// TIA Portal project "myproject" (V16)

(* hardware
DEVICE "S71500/ET200MP-Station_1"  S7-1500 station
   slot 0: "Profilschiene_0"  6ES7 590-1***0-0AA0
   slot 1: "PLC_1"  CPU 1511-1 PN  6ES7 511-1AK00-0AB0  V1.8
   slot 2: "AI 8xU/I/RTD/TC ST_1"  AI 8xU/I/RTD/TC ST  6ES7 531-7KF00-0AB0  V2.0
   slot 3: "AI 8xU/I/RTD/TC ST_2"  AI 8xU/I/RTD/TC ST  6ES7 531-7KF00-0AB0  V2.0
   slot 4: "AI 8xU/I/RTD/TC ST_3"  AI 8xU/I/RTD/TC ST  6ES7 531-7KF00-0AB0  V2.0
   slot 5: "AI 8xU/I/RTD/TC ST_4"  AI 8xU/I/RTD/TC ST  6ES7 531-7KF00-0AB0  V2.0
   slot 6: "DI 16x24VDC BA_1"  DI 16x24VDC BA  6ES7 521-1BH10-0AA0  V1.0
   slot 7: "DI 16x24VDC / DQ 16x24VDC/0.5A BA_1"  DI 16x24VDC/DQ 16x24VDC/0.5A BA  6ES7 523-1BL00-0AA0  V1.1
   slot 8: "DI 16x24VDC / DQ 16x24VDC/0.5A BA_2"  DI 16x24VDC/DQ 16x24VDC/0.5A BA  6ES7 523-1BL00-0AA0  V1.1
DEVICE "HMI_1"  TP700 Comfort INOX PCT
   slot 0: "HMI_1"  TP700 Comfort INOX PCT  6AV2 144-8GC20-0AA0  16.0.0.0
   slot 1: "HMI_RT_1"  TP700 Comfort INOX PCT  6AV2 144-8GC20-0AA0  16.0.0.0
   slot 5: "HMI_1.IE_CP_1"  PROFINET Interface  16.0.0.0
      slot 1: "PROFINET Interface_1"  PROFINET Interface
         slot 1: "Port_1"  Port
         slot 2: "Port_2"  Port
   slot 7: "HMI_1.MPI/DP_CP_1"  MPI/DP Interface  16.0.0.0
*)

// ===== PLC "PLC_1"  CPU 1511-1 PN =====

VAR_GLOBAL   // PLC tag table "Standard-Variablentabelle"
   "compteur_boites" AT %C1 : Counter;
   "compteur_bouteilles" AT %C2 : Counter;
   "tag11" AT %M6.1 : Bool;
END_VAR

VAR_GLOBAL   // PLC tag table "Input/output"
   "c1" AT %I0.0 : Bool;   // capteur plastique fondu
   "mc1" AT %Q0.0 : Bool;   // moteur convoyeur 1
   "cm1" AT %I0.1 : Bool;   // capteur devant machine 1
   "m1" AT %Q0.1 : Bool;   // moteur machine moulage
   "cm11" AT %I0.2 : Bool;   // capteur apres machine moulage
   "mc2" AT %Q0.2 : Bool;   // moteur convoyeur 2
   "mcb" AT %Q0.3 : Bool;   // moteur curved belt
   "cl" AT %I0.3 : Bool;   // capteur boite
   "lids conveyor" AT %Q0.4 : Bool;   // convoyeur boite-assemblage
   "base conveyor" AT %Q0.5 : Bool;   // convoyeur base-assemblage
   "lid clamped" AT %I0.4 : Bool;   // clamped boite
   "base clamped" AT %I0.5 : Bool;   // clamped base
   "clamp lid" AT %Q0.6 : Bool;   // clamper la boite
   "clamp base" AT %Q0.7 : Bool;   // clamper la base
   "move x assemb" AT %Q1.0 : Bool;   // translation m. assemblage sur x
   "move z assemb" AT %Q1.1 : Bool;   // translation m. assemblage sur z
   "moved x assemb" AT %I0.6 : Bool;   // translation en cours sur x
   "moved z assemb" AT %I0.7 : Bool;   // translation en cours sur z
   "raise assemb" AT %Q1.2 : Bool;   // relever la barre devant produit assemblé
   "grab assemb" AT %Q1.3 : Bool;   // grab de la boite
   "grabbed assemb" AT %I1.4 : Bool;   // boite grabbed
   "lid at place" AT %I1.0 : Bool;   // boite en place
   "base at place" AT %I1.1 : Bool;   // base en place
   "part leaving" AT %I1.2 : Bool;   // piece sortante
   "cc" AT %I1.3 : Bool;   // capteur bol
   "ettiquetage conveyor" AT %Q1.5 : Bool;   // convoyeur ettiquette
   "product conveyor" AT %Q1.6 : Bool;   // convoyeur bol/ettiquetage
   "box clamped" AT %I2.7 : Bool;   // clamped ett
   "product clamped" AT %I1.5 : Bool;   // clamped bol/ettiquetage
   "clamp ettiquete" AT %Q1.7 : Bool;   // clamper l'ettiquette
   "clamp product" AT %Q2.0 : Bool;   // clamper le bol/ettiquetage
   "move x ett" AT %Q2.1 : Bool;   // translation m. etti sur x
   "move z ett" AT %Q2.2 : Bool;   // translation m. etti sur z
   "moved x ett" AT %I1.6 : Bool;   // translation en cours sur x
   "moved z ett" AT %I1.7 : Bool;   // translation en cours sur z
   "raise ett" AT %Q2.3 : Bool;   // relever la barre devant produit etti
   "grab ett" AT %Q2.4 : Bool;   // grab du produit
   "grabbed ett" AT %I3.1 : Bool;   // produit grabbed
   "ettiquete at place" AT %I2.0 : Bool;   // ettiquete en place
   "product at place" AT %I2.1 : Bool;   // produit en place
   "product leaving" AT %I2.2 : Bool;   // produit sortant
   "dcy" AT %I2.3 : Bool;   // bouton debut cycle
   "fcy" AT %I2.4 : Bool;   // bouton fin cycle
   "au" AT %I2.5 : Bool;   // bouton urgence
   "emetteur plastique" AT %Q2.6 : Bool;   // emetteur plastique fondu
   "emetteur base" AT %Q2.7 : Bool;   // emetteur base du jouet
   "emetteur bol" AT %Q3.0 : Bool;   // emetteur carton d'emballage
   "emetteur ettiquete" AT %Q3.1 : Bool;   // emetteur box d'emballage
   "tag1" AT %M3.2 : Bool;
   "tag2" AT %M3.3 : Bool;
   "tag3" AT %M3.4 : Bool;
   "tag4" AT %M3.5 : Bool;
   "cp" AT %I3.0 : Bool;   // capteur piece assemblée
   "raised assembly" AT %I3.2 : Bool;   // barre raised assembly
   "raised ettiq" AT %I3.3 : Bool;   // barre raised ett
   "bol conveyor" AT %Q3.2 : Bool;   // convoyeur des bols
   "cp2" AT %I3.4 : Bool;   // capteur piece assemblée sortante
   "cb" AT %I3.5 : Bool;   // capteur ettiquette
   "cp3" AT %I3.6 : Bool;   // capteur produit ettiqueté
   "tag5" AT %M3.7 : Bool;
   "tag6" AT %M4.0 : Bool;
   "tag7" AT %M4.1 : Bool;
   "tag8" AT %M4.2 : Bool;
   "remover" AT %Q3.3 : Bool;   // stock de sortie
   "tag9" AT %M5.7 : Bool;
   "vv" AT %Q3.4 : Bool;   // voyant vert de marche du systeme
   "vo" AT %Q3.5 : Bool;   // voyant orangé d'arret fin de cycle
   "vr" AT %Q3.6 : Bool;   // voyant rouge d'arret d'urgence
   "tag10" AT %M6.0 : Bool;
END_VAR

// folder: System blocks/Program resources

DATA_BLOCK "tp move z"   // DB1
{ S7_Optimized_Access := 'TRUE' }
AUTHOR : Simatic
FAMILY : IEC
NAME : IEC_TMR
VERSION : 1.0
// stored: InstanceOfName IEC_TIMER
"IEC_TIMER"
BEGIN
END_DATA_BLOCK

DATA_BLOCK "timer3"   // DB2
{ S7_Optimized_Access := 'TRUE' }
AUTHOR : Simatic
FAMILY : IEC
NAME : IEC_TMR
VERSION : 1.0
// stored: InstanceOfName IEC_TIMER
"IEC_TIMER"
BEGIN
END_DATA_BLOCK

DATA_BLOCK "time1"   // DB3
{ S7_Optimized_Access := 'TRUE' }
AUTHOR : Simatic
FAMILY : IEC
NAME : IEC_TMR
VERSION : 1.0
// stored: InstanceOfName IEC_TIMER
"IEC_TIMER"
BEGIN
END_DATA_BLOCK

DATA_BLOCK "timer4"   // DB4
{ S7_Optimized_Access := 'TRUE' }
AUTHOR : Simatic
FAMILY : IEC
NAME : IEC_TMR
VERSION : 1.0
// stored: InstanceOfName IEC_TIMER
"IEC_TIMER"
BEGIN
END_DATA_BLOCK

DATA_BLOCK "counter_boites"   // DB5
{ S7_Optimized_Access := 'TRUE' }
AUTHOR : Simatic
FAMILY : IEC
NAME : CNTR
VERSION : 1.0
// stored: InstanceOfName IEC_COUNTER
"IEC_COUNTER"
BEGIN
END_DATA_BLOCK

DATA_BLOCK "counter_bols"   // DB6
{ S7_Optimized_Access := 'TRUE' }
AUTHOR : Simatic
FAMILY : IEC
NAME : CNTR
VERSION : 1.0
// stored: InstanceOfName IEC_COUNTER
"IEC_COUNTER"
BEGIN
END_DATA_BLOCK

// folder: (top level)

FUNCTION "MHJ-PLC-Lab-Function-S71500" : Void   // FC9000, SCL
{ S7_Optimized_Access := 'TRUE' }
VERSION : 0.1
   VAR_TEMP
      Value : Byte;
      ForCounter : Int;
   END_VAR
   VAR CONSTANT
      Value_01_DW : DWord := 16#1223_5486;
      Value_02_DW : DWord := 16#A6C9_D1F5;
   END_VAR
BEGIN

   #Value:=PEEK(area := 16#82,
        dbNumber := 0,
        byteOffset := 511);
   #Value := #Value + 1;

   POKE(area := 16#82,
        dbNumber := 0,
        byteOffset := 511,
        value := #Value);

   POKE(area := 16#82,
        dbNumber := 0,
        byteOffset := 1016,
        value := #Value_01_DW);
   POKE(area := 16#82,
        dbNumber := 0,
        byteOffset := 1020,
        value := #Value_02_DW);

   FOR #ForCounter := 0 TO 63 DO
       #Value:=PEEK(area := 16#1,
            dbNumber := 0,
            byteOffset := #ForCounter);
       POKE(area := 16#81,
            dbNumber := 0,
            byteOffset := #ForCounter,
            value := #Value);
   END_FOR;
   #Value := PEEK(area := 16#1,
                  dbNumber := 0,
                  byteOffset := 512);
   POKE(area := 16#82,
        dbNumber := 0,
        byteOffset := 512,
        value := #Value);
END_FUNCTION

ORGANIZATION_BLOCK "Main"   // OB1, LAD, ProgramCycle
TITLE = "Main Program Sweep (Cycle)"
{ S7_Optimized_Access := 'TRUE' }
VERSION : 0.1
   VAR_INPUT
      Initial_Call : Bool;   // Initial call of this OB
      Remanence : Bool;   // =True, if remanent data are available
   END_VAR
   VAR_TEMP   // added for the SCL form of the ladder/FBD networks
      _w1 : Bool;
      _w2 : Bool;
   END_VAR
BEGIN

REGION Network 1
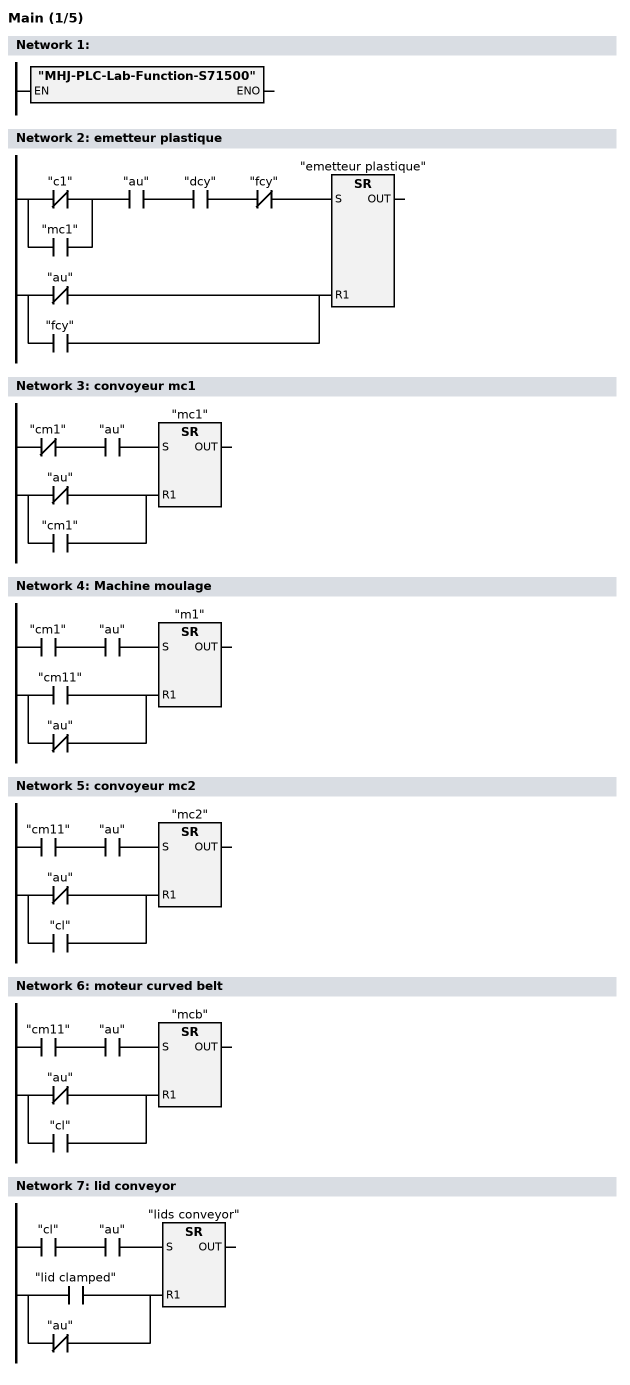
   RUNG wire#powerrail
      "MHJ-PLC-Lab-Function-S71500"()
   END_RUNG
   // the same network as SCL:
   "MHJ-PLC-Lab-Function-S71500"();
END_REGION

REGION Network 2: emetteur plastique
   RUNG wire#powerrail
      I_Contact( "c1" )
      wire#w1
      Contact( "au" )
      Contact( "dcy" )
      I_Contact( "fcy" )
      S_SR(operand := "emetteur plastique", r1 := wire#w2)
   END_RUNG
   RUNG wire#powerrail
      Contact( "mc1" )
   END_RUNG wire#w1
   RUNG wire#powerrail
      I_Contact( "au" )
   END_RUNG wire#w2
   RUNG wire#powerrail
      Contact( "fcy" )
   END_RUNG wire#w2
   // the same network as SCL:
   IF (NOT "c1" OR "mc1") AND "au" AND "dcy" AND NOT "fcy" THEN
       "emetteur plastique" := TRUE;   // SR flip-flop
   END_IF;
   IF NOT "au" OR "fcy" THEN "emetteur plastique" := FALSE; END_IF;
END_REGION

REGION Network 3: convoyeur mc1
   RUNG wire#powerrail
      I_Contact( "cm1" )
      Contact( "au" )
      S_SR(operand := "mc1", r1 := wire#w1)
   END_RUNG
   RUNG wire#powerrail
      I_Contact( "au" )
   END_RUNG wire#w1
   RUNG wire#powerrail
      Contact( "cm1" )
   END_RUNG wire#w1
   // the same network as SCL:
   IF NOT "cm1" AND "au" THEN
       "mc1" := TRUE;   // SR flip-flop
   END_IF;
   IF NOT "au" OR "cm1" THEN "mc1" := FALSE; END_IF;
END_REGION

REGION Network 4: Machine moulage
   RUNG wire#powerrail
      Contact( "cm1" )
      Contact( "au" )
      S_SR(operand := "m1", r1 := wire#w1)
   END_RUNG
   RUNG wire#powerrail
      Contact( "cm11" )
   END_RUNG wire#w1
   RUNG wire#powerrail
      I_Contact( "au" )
   END_RUNG wire#w1
   // the same network as SCL:
   IF "cm1" AND "au" THEN
       "m1" := TRUE;   // SR flip-flop
   END_IF;
   IF "cm11" OR NOT "au" THEN "m1" := FALSE; END_IF;
END_REGION

REGION Network 5: convoyeur mc2
   RUNG wire#powerrail
      Contact( "cm11" )
      Contact( "au" )
      S_SR(operand := "mc2", r1 := wire#w1)
   END_RUNG
   RUNG wire#powerrail
      I_Contact( "au" )
   END_RUNG wire#w1
   RUNG wire#powerrail
      Contact( "cl" )
   END_RUNG wire#w1
   // the same network as SCL:
   IF "cm11" AND "au" THEN
       "mc2" := TRUE;   // SR flip-flop
   END_IF;
   IF NOT "au" OR "cl" THEN "mc2" := FALSE; END_IF;
END_REGION

REGION Network 6: moteur curved belt
   RUNG wire#powerrail
      Contact( "cm11" )
      Contact( "au" )
      S_SR(operand := "mcb", r1 := wire#w1)
   END_RUNG
   RUNG wire#powerrail
      I_Contact( "au" )
   END_RUNG wire#w1
   RUNG wire#powerrail
      Contact( "cl" )
   END_RUNG wire#w1
   // the same network as SCL:
   IF "cm11" AND "au" THEN
       "mcb" := TRUE;   // SR flip-flop
   END_IF;
   IF NOT "au" OR "cl" THEN "mcb" := FALSE; END_IF;
END_REGION

REGION Network 7: lid conveyor
   RUNG wire#powerrail
      Contact( "cl" )
      Contact( "au" )
      S_SR(operand := "lids conveyor", r1 := wire#w1)
   END_RUNG
   RUNG wire#powerrail
      Contact( "lid clamped" )
   END_RUNG wire#w1
   RUNG wire#powerrail
      I_Contact( "au" )
   END_RUNG wire#w1
   // the same network as SCL:
   IF "cl" AND "au" THEN
       "lids conveyor" := TRUE;   // SR flip-flop
   END_IF;
   IF "lid clamped" OR NOT "au" THEN "lids conveyor" := FALSE; END_IF;
END_REGION

REGION Network 8: clamping lid
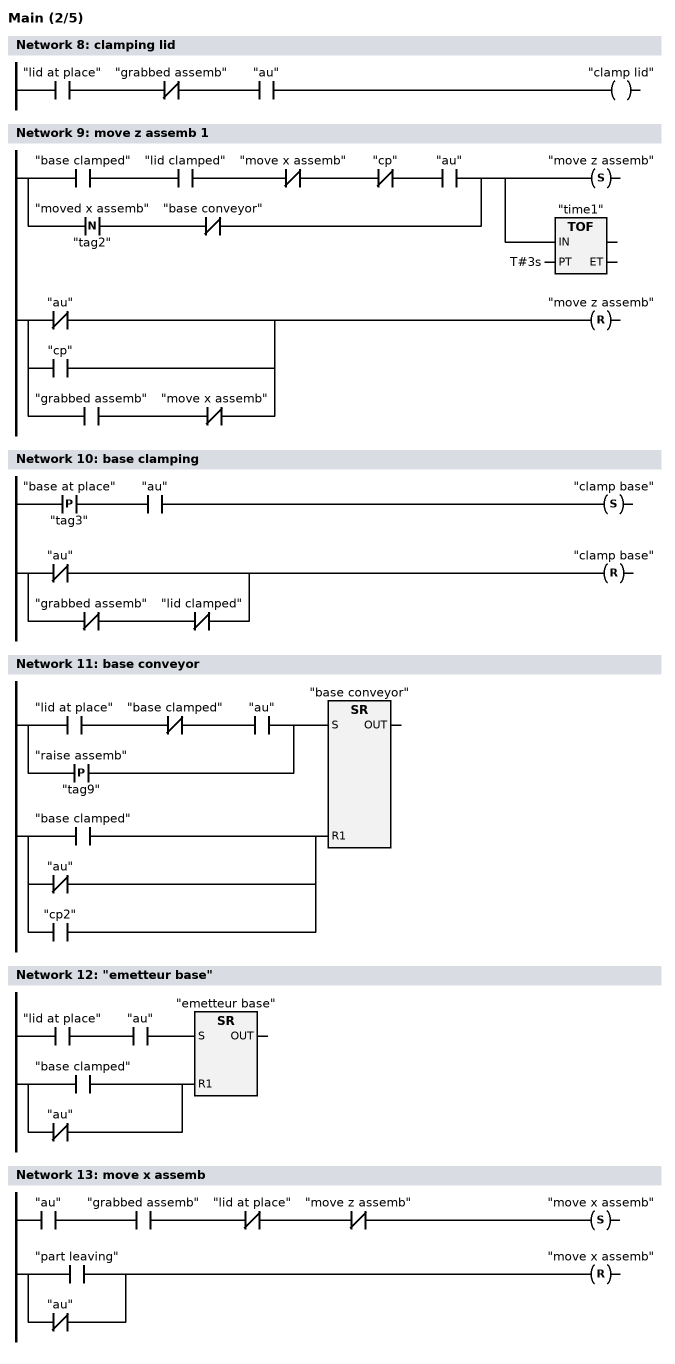
   RUNG wire#powerrail
      Contact( "lid at place" )
      I_Contact( "grabbed assemb" )
      Contact( "au" )
      Coil( "clamp lid" )
   END_RUNG
   // the same network as SCL:
   "clamp lid" := "lid at place" AND NOT "grabbed assemb" AND "au";
END_REGION

REGION Network 9: move z assemb 1
   #_w1 := NOT "moved x assemb" AND "tag2";   // falling edge of "moved x assemb"
   "tag2" := "moved x assemb";
   #_w2 := ("base clamped" AND "lid clamped" AND NOT "move x assemb" AND NOT "cp" AND "au") OR (#_w1 AND NOT "base conveyor");
   IF #_w2 THEN "move z assemb" := TRUE; END_IF;
   "time1".TOF(IN := #_w2, PT := T#3s);
   IF NOT "au" OR "cp" OR ("grabbed assemb" AND NOT "move x assemb") THEN "move z assemb" := FALSE; END_IF;
END_REGION

REGION Network 10: base clamping
   RUNG wire#powerrail
      P_Contact(operand := "base at place", bit := "tag3")
      Contact( "au" )
      S_Coil( "clamp base" )
   END_RUNG
   RUNG wire#powerrail
      I_Contact( "au" )
      wire#w1
      R_Coil( "clamp base" )
   END_RUNG
   RUNG wire#powerrail
      I_Contact( "grabbed assemb" )
      I_Contact( "lid clamped" )
   END_RUNG wire#w1
   // the same network as SCL:
   #_w1 := "base at place" AND NOT "tag3";   // rising edge of "base at place"
   "tag3" := "base at place";
   IF #_w1 AND "au" THEN "clamp base" := TRUE; END_IF;
   IF NOT "au" OR (NOT "grabbed assemb" AND NOT "lid clamped") THEN "clamp base" := FALSE; END_IF;
END_REGION

REGION Network 11: base conveyor
   RUNG wire#powerrail
      Contact( "lid at place" )
      I_Contact( "base clamped" )
      Contact( "au" )
      wire#w1
      S_SR(operand := "base conveyor", r1 := wire#w2)
   END_RUNG
   RUNG wire#powerrail
      P_Contact(operand := "raise assemb", bit := "tag9")
   END_RUNG wire#w1
   RUNG wire#powerrail
      Contact( "base clamped" )
   END_RUNG wire#w2
   RUNG wire#powerrail
      I_Contact( "au" )
   END_RUNG wire#w2
   RUNG wire#powerrail
      Contact( "cp2" )
   END_RUNG wire#w2
   // the same network as SCL:
   #_w1 := "raise assemb" AND NOT "tag9";   // rising edge of "raise assemb"
   "tag9" := "raise assemb";
   IF ("lid at place" AND NOT "base clamped" AND "au") OR #_w1 THEN
       "base conveyor" := TRUE;   // SR flip-flop
   END_IF;
   IF "base clamped" OR NOT "au" OR "cp2" THEN "base conveyor" := FALSE; END_IF;
END_REGION

REGION Network 12: "emetteur base"
   RUNG wire#powerrail
      Contact( "lid at place" )
      Contact( "au" )
      S_SR(operand := "emetteur base", r1 := wire#w1)
   END_RUNG
   RUNG wire#powerrail
      Contact( "base clamped" )
   END_RUNG wire#w1
   RUNG wire#powerrail
      I_Contact( "au" )
   END_RUNG wire#w1
   // the same network as SCL:
   IF "lid at place" AND "au" THEN
       "emetteur base" := TRUE;   // SR flip-flop
   END_IF;
   IF "base clamped" OR NOT "au" THEN "emetteur base" := FALSE; END_IF;
END_REGION

REGION Network 13: move x assemb
   RUNG wire#powerrail
      Contact( "au" )
      Contact( "grabbed assemb" )
      I_Contact( "lid at place" )
      I_Contact( "move z assemb" )
      S_Coil( "move x assemb" )
   END_RUNG
   RUNG wire#powerrail
      Contact( "part leaving" )
      wire#w1
      R_Coil( "move x assemb" )
   END_RUNG
   RUNG wire#powerrail
      I_Contact( "au" )
   END_RUNG wire#w1
   // the same network as SCL:
   IF "au" AND "grabbed assemb" AND NOT "lid at place" AND NOT "move z assemb" THEN
       "move x assemb" := TRUE;
   END_IF;
   IF "part leaving" OR NOT "au" THEN "move x assemb" := FALSE; END_IF;
END_REGION

REGION Network 14: grab assem
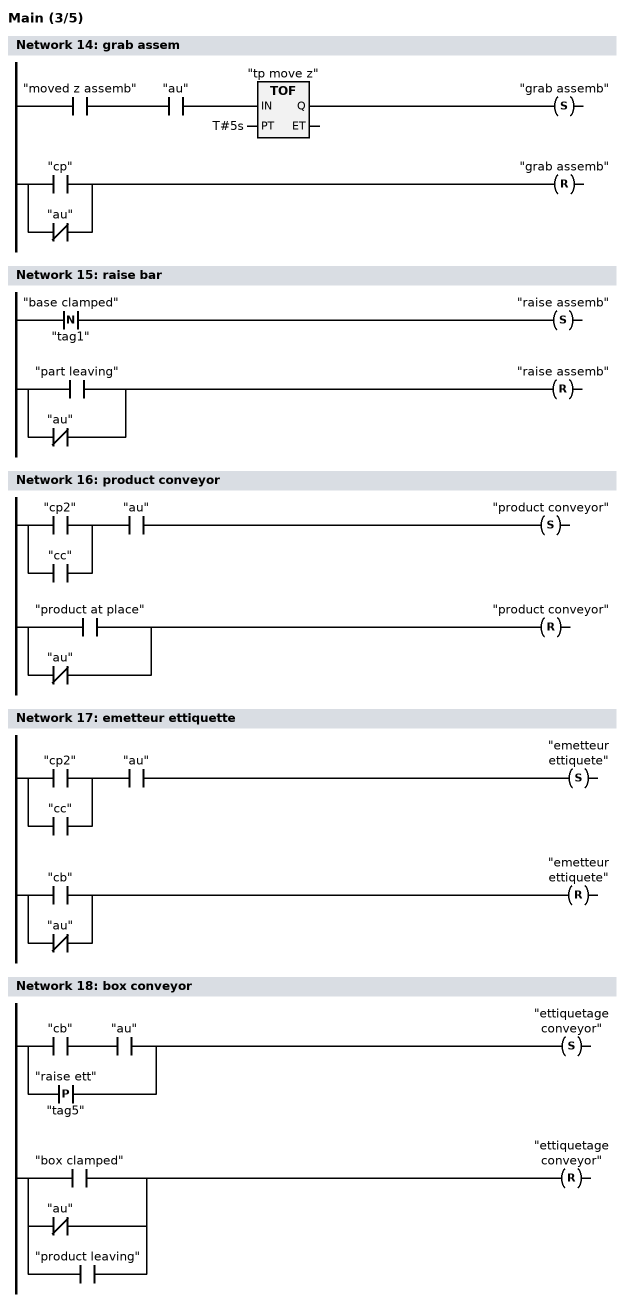
   "tp move z".TOF(IN := "moved z assemb" AND "au", PT := T#5s);
   IF "tp move z".Q THEN "grab assemb" := TRUE; END_IF;
   IF "cp" OR NOT "au" THEN "grab assemb" := FALSE; END_IF;
END_REGION

REGION Network 15: raise bar
   RUNG wire#powerrail
      N_Contact(operand := "base clamped", bit := "tag1")
      S_Coil( "raise assemb" )
   END_RUNG
   RUNG wire#powerrail
      Contact( "part leaving" )
      wire#w1
      R_Coil( "raise assemb" )
   END_RUNG
   RUNG wire#powerrail
      I_Contact( "au" )
   END_RUNG wire#w1
   // the same network as SCL:
   #_w1 := NOT "base clamped" AND "tag1";   // falling edge of "base clamped"
   "tag1" := "base clamped";
   IF #_w1 THEN "raise assemb" := TRUE; END_IF;
   IF "part leaving" OR NOT "au" THEN "raise assemb" := FALSE; END_IF;
END_REGION

REGION Network 16: product conveyor
   RUNG wire#powerrail
      Contact( "cp2" )
      wire#w1
      Contact( "au" )
      S_Coil( "product conveyor" )
   END_RUNG
   RUNG wire#powerrail
      Contact( "cc" )
   END_RUNG wire#w1
   RUNG wire#powerrail
      Contact( "product at place" )
      wire#w2
      R_Coil( "product conveyor" )
   END_RUNG
   RUNG wire#powerrail
      I_Contact( "au" )
   END_RUNG wire#w2
   // the same network as SCL:
   IF ("cp2" OR "cc") AND "au" THEN "product conveyor" := TRUE; END_IF;
   IF "product at place" OR NOT "au" THEN "product conveyor" := FALSE; END_IF;
END_REGION

REGION Network 17: emetteur ettiquette
   RUNG wire#powerrail
      Contact( "cp2" )
      wire#w1
      Contact( "au" )
      S_Coil( "emetteur ettiquete" )
   END_RUNG
   RUNG wire#powerrail
      Contact( "cc" )
   END_RUNG wire#w1
   RUNG wire#powerrail
      Contact( "cb" )
      wire#w2
      R_Coil( "emetteur ettiquete" )
   END_RUNG
   RUNG wire#powerrail
      I_Contact( "au" )
   END_RUNG wire#w2
   // the same network as SCL:
   IF ("cp2" OR "cc") AND "au" THEN "emetteur ettiquete" := TRUE; END_IF;
   IF "cb" OR NOT "au" THEN "emetteur ettiquete" := FALSE; END_IF;
END_REGION

REGION Network 18: box conveyor
   RUNG wire#powerrail
      Contact( "cb" )
      Contact( "au" )
      wire#w1
      S_Coil( "ettiquetage conveyor" )
   END_RUNG
   RUNG wire#powerrail
      P_Contact(operand := "raise ett", bit := "tag5")
   END_RUNG wire#w1
   RUNG wire#powerrail
      Contact( "box clamped" )
      wire#w2
      R_Coil( "ettiquetage conveyor" )
   END_RUNG
   RUNG wire#powerrail
      I_Contact( "au" )
   END_RUNG wire#w2
   RUNG wire#powerrail
      Contact( "product leaving" )
   END_RUNG wire#w2
   // the same network as SCL:
   #_w1 := "raise ett" AND NOT "tag5";   // rising edge of "raise ett"
   "tag5" := "raise ett";
   IF ("cb" AND "au") OR #_w1 THEN "ettiquetage conveyor" := TRUE; END_IF;
   IF "box clamped" OR NOT "au" OR "product leaving" THEN "ettiquetage conveyor" := FALSE; END_IF;
END_REGION

REGION Network 19: emetteur bol
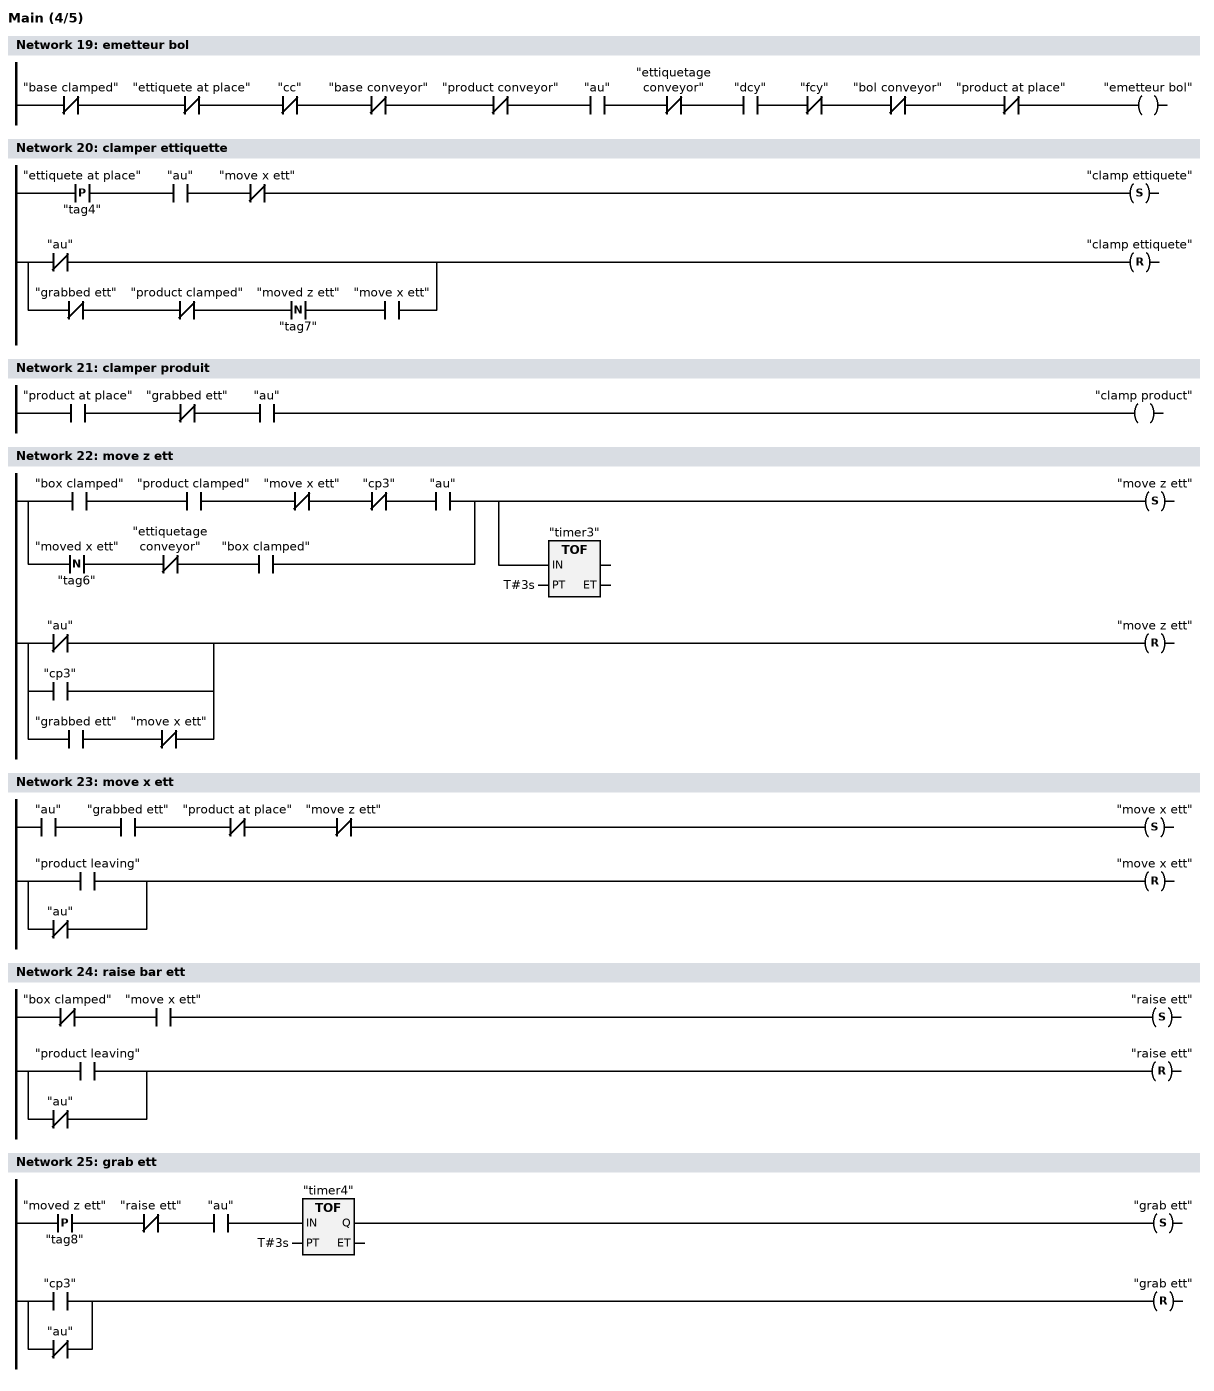
   RUNG wire#powerrail
      I_Contact( "base clamped" )
      I_Contact( "ettiquete at place" )
      I_Contact( "cc" )
      I_Contact( "base conveyor" )
      I_Contact( "product conveyor" )
      Contact( "au" )
      I_Contact( "ettiquetage conveyor" )
      Contact( "dcy" )
      I_Contact( "fcy" )
      I_Contact( "bol conveyor" )
      I_Contact( "product at place" )
      Coil( "emetteur bol" )
   END_RUNG
   // the same network as SCL:
   "emetteur bol" := NOT "base clamped" AND NOT "ettiquete at place" AND NOT "cc" AND NOT "base conveyor" AND NOT "product conveyor" AND "au" AND NOT "ettiquetage conveyor" AND "dcy" AND NOT "fcy" AND NOT "bol conveyor" AND NOT "product at place";
END_REGION

REGION Network 20: clamper ettiquette
   RUNG wire#powerrail
      P_Contact(operand := "ettiquete at place", bit := "tag4")
      Contact( "au" )
      I_Contact( "move x ett" )
      S_Coil( "clamp ettiquete" )
   END_RUNG
   RUNG wire#powerrail
      I_Contact( "au" )
      wire#w1
      R_Coil( "clamp ettiquete" )
   END_RUNG
   RUNG wire#powerrail
      I_Contact( "grabbed ett" )
      I_Contact( "product clamped" )
      N_Contact(operand := "moved z ett", bit := "tag7")
      Contact( "move x ett" )
   END_RUNG wire#w1
   // the same network as SCL:
   #_w1 := "ettiquete at place" AND NOT "tag4";   // rising edge of "ettiquete at place"
   "tag4" := "ettiquete at place";
   IF #_w1 AND "au" AND NOT "move x ett" THEN "clamp ettiquete" := TRUE; END_IF;
   #_w2 := NOT "grabbed ett" AND NOT "product clamped" AND NOT "moved z ett" AND "tag7";   // falling edge of "moved z ett"
   "tag7" := "moved z ett";
   IF NOT "au" OR (#_w2 AND "move x ett") THEN "clamp ettiquete" := FALSE; END_IF;
END_REGION

REGION Network 21: clamper produit
   RUNG wire#powerrail
      Contact( "product at place" )
      I_Contact( "grabbed ett" )
      Contact( "au" )
      Coil( "clamp product" )
   END_RUNG
   // the same network as SCL:
   "clamp product" := "product at place" AND NOT "grabbed ett" AND "au";
END_REGION

REGION Network 22: move z ett
   #_w1 := NOT "moved x ett" AND "tag6";   // falling edge of "moved x ett"
   "tag6" := "moved x ett";
   #_w2 := ("box clamped" AND "product clamped" AND NOT "move x ett" AND NOT "cp3" AND "au") OR (#_w1 AND NOT "ettiquetage conveyor" AND "box clamped");
   IF #_w2 THEN "move z ett" := TRUE; END_IF;
   "timer3".TOF(IN := #_w2, PT := T#3s);
   IF NOT "au" OR "cp3" OR ("grabbed ett" AND NOT "move x ett") THEN "move z ett" := FALSE; END_IF;
END_REGION

REGION Network 23: move x ett
   RUNG wire#powerrail
      Contact( "au" )
      Contact( "grabbed ett" )
      I_Contact( "product at place" )
      I_Contact( "move z ett" )
      S_Coil( "move x ett" )
   END_RUNG
   RUNG wire#powerrail
      Contact( "product leaving" )
      wire#w1
      R_Coil( "move x ett" )
   END_RUNG
   RUNG wire#powerrail
      I_Contact( "au" )
   END_RUNG wire#w1
   // the same network as SCL:
   IF "au" AND "grabbed ett" AND NOT "product at place" AND NOT "move z ett" THEN
       "move x ett" := TRUE;
   END_IF;
   IF "product leaving" OR NOT "au" THEN "move x ett" := FALSE; END_IF;
END_REGION

REGION Network 24: raise bar ett
   RUNG wire#powerrail
      I_Contact( "box clamped" )
      Contact( "move x ett" )
      S_Coil( "raise ett" )
   END_RUNG
   RUNG wire#powerrail
      Contact( "product leaving" )
      wire#w1
      R_Coil( "raise ett" )
   END_RUNG
   RUNG wire#powerrail
      I_Contact( "au" )
   END_RUNG wire#w1
   // the same network as SCL:
   IF NOT "box clamped" AND "move x ett" THEN "raise ett" := TRUE; END_IF;
   IF "product leaving" OR NOT "au" THEN "raise ett" := FALSE; END_IF;
END_REGION

REGION Network 25: grab ett
   #_w1 := "moved z ett" AND NOT "tag8";   // rising edge of "moved z ett"
   "tag8" := "moved z ett";
   "timer4".TOF(IN := #_w1 AND NOT "raise ett" AND "au", PT := T#3s);
   IF "timer4".Q THEN "grab ett" := TRUE; END_IF;
   IF "cp3" OR NOT "au" THEN "grab ett" := FALSE; END_IF;
END_REGION

REGION Network 26: remover
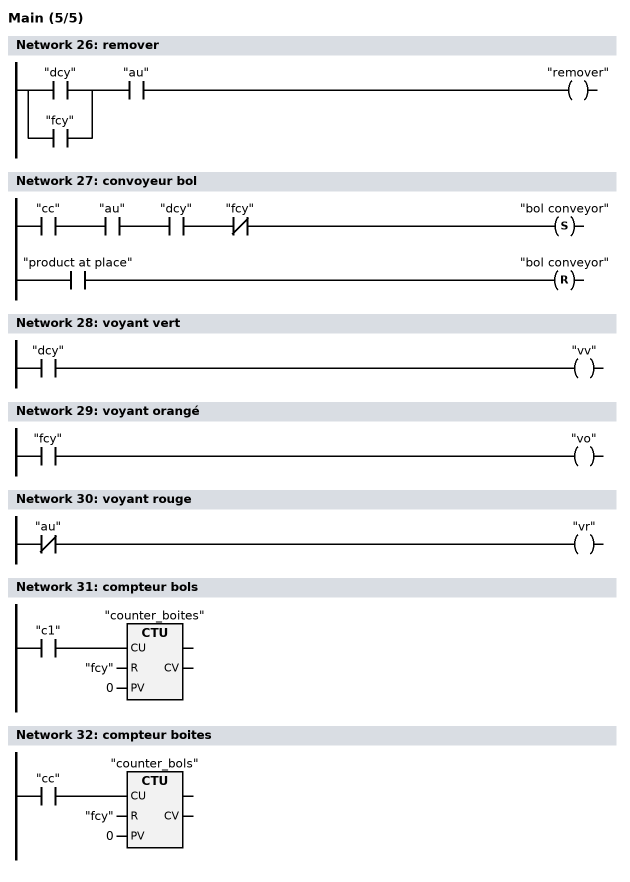
   RUNG wire#powerrail
      Contact( "dcy" )
      wire#w1
      Contact( "au" )
      Coil( "remover" )
   END_RUNG
   RUNG wire#powerrail
      Contact( "fcy" )
   END_RUNG wire#w1
   // the same network as SCL:
   "remover" := ("dcy" OR "fcy") AND "au";
END_REGION

REGION Network 27: convoyeur bol
   RUNG wire#powerrail
      Contact( "cc" )
      Contact( "au" )
      Contact( "dcy" )
      I_Contact( "fcy" )
      S_Coil( "bol conveyor" )
   END_RUNG
   RUNG wire#powerrail
      Contact( "product at place" )
      R_Coil( "bol conveyor" )
   END_RUNG
   // the same network as SCL:
   IF "cc" AND "au" AND "dcy" AND NOT "fcy" THEN "bol conveyor" := TRUE; END_IF;
   IF "product at place" THEN "bol conveyor" := FALSE; END_IF;
END_REGION

REGION Network 28: voyant vert
   RUNG wire#powerrail
      Contact( "dcy" )
      Coil( "vv" )
   END_RUNG
   // the same network as SCL:
   "vv" := "dcy";
END_REGION

REGION Network 29: voyant orangé
   RUNG wire#powerrail
      Contact( "fcy" )
      Coil( "vo" )
   END_RUNG
   // the same network as SCL:
   "vo" := "fcy";
END_REGION

REGION Network 30: voyant rouge
   RUNG wire#powerrail
      I_Contact( "au" )
      Coil( "vr" )
   END_RUNG
   // the same network as SCL:
   "vr" := NOT "au";
END_REGION

REGION Network 31: compteur bols
   "counter_boites".CTU(CU := "c1", R := "fcy", PV := 0);
END_REGION

REGION Network 32: compteur boites
   "counter_bols".CTU(CU := "cc", R := "fcy", PV := 0);
END_REGION
END_ORGANIZATION_BLOCK

(* ===== HMI "HMI_RT_1" =====
system functions are stored by id; their names below are inferred from use
connection "HMI_Connection_1": ETHERNET, S7_1500_OMS

HMI tags "Default tag table"
   "dcy" : Bool = PLC dcy AT %I2.3, 1 s
   "fcy" : Bool = PLC fcy AT %I2.4, 1 s
   "au" : Bool = PLC au AT %I2.5, 1 s
   "cv_boites" : Int = PLC counter_boites.CV AT %DB1.DBX0.0, 1 s
   "cv_bouteilles" : Int = PLC counter_bols.CV AT %DB1.DBW0, 1 s

screen "Screen_1" 800x480
   GraphicIOField "PlotLight_Round_N_Mono" at 0,76 size 50x50; PictureOff "PilotLight_Round_N_On_mono"; PictureOn "PilotLight_Round_N_Off_mono"
      Appearance <- "dcy"
      ProcessValue <- "dcy"
   GraphicIOField "PlotLight_Round_G" at 0,164 size 50x50; PictureOn "PilotLight_Round_G_On_256c"; PictureOff "PilotLight_Round_G_Off_256c"
      Appearance <- "dcy"
      ProcessValue <- "dcy"
   GraphicIOField "PlotLight_Round_R" at 0,4 size 50x50; PictureOn "PilotLight_Round_R_On_256c"; PictureOff "PilotLight_Round_R_Off_256c"
      ProcessValue <- "au"
      Appearance <- "au"
      ObjectEnable <- "au"
   IOField "I/O field_2" at 108,288 size 198x55; FormatPattern s99999
      ProcessValue <- "cv_boites"
   Switch "Pushbutton_Emergency" at 125,1 size 80x80; CaptionText 'Switch'; TextOff '0'; TextOn '1'; PictureOff "Pushbutton_Emergency_Off_256c"; PictureOn "Pushbutton_Emergency_On_256c"
      on SwitchOn: SetBit("au")
      on SwitchOff: ResetBit("au")
      ProcessValue <- "au"
   IOField "I/O field_1" at 523,289 size 198x55; FormatPattern s99999
      ProcessValue <- "cv_bouteilles"
   TextField "Text field_1" at 83,252 size 275x23; Text 'Boites assemblees étiquetées'
   TextField "Text field_2" at 557,254 size 135x23; Text 'Bols étiquetés'
   Switch "Toggle_Vertical_G" at 147,114 size 50x80; CaptionText 'Switch'; TextOff '0'; TextOn '1'; PictureOff "Toggle_Vertical_G_Off_256c"; PictureOn "Toggle_Vertical_G_On_256c"
      ProcessValue <- "dcy"
      Appearance <- "dcy"
   TextField "Text field_4" at 208,132 size 42x23; Text 'DCY'
   TextField "Text field_5" at 208,164 size 39x23; Text 'FCY'
   TextField "Text field_3" at 228,31 size 183x23; Text 'ARRET D'URGENCE'
*)